// TwinCAT 3 PLC project SPS
// Company: mbc engineering GmbH
// ProgramVersion: 3.1.4022.2
// libraries:
//   Tc2_Standard, * (Beckhoff Automation GmbH)
//   Tc2_System, * (Beckhoff Automation GmbH)
//   Tc3_Module, * (Beckhoff Automation GmbH)
//   MBC TC3 PCS Library,newest,mbc engineering GmbH
// project tree:
//   Commands/ AddCommand.TcPOU, Commands.TcGVL, CustomStateCommand.TcPOU, DelayedAddCommand.TcPOU, FB_CommandWithStruct.TcPOU, PRG_Commands.TcPOU, TriggerCommand.TcPOU
//   DUTs/ E_EnumType.TcDUT, ST_CommandArgs.TcDUT
//   / PlcTask.TcTTO (not stored)
//   POUs/ MAIN.TcPOU

// ---- DUTs/E_EnumType.TcDUT
{attribute 'qualified_only'}
{attribute 'strict'}
TYPE E_EnumType :
(
	eValue0 := 0,
	eValue1 := 1,
	eValue2 := 3
);
END_TYPE

// ---- DUTs/ST_CommandArgs.TcDUT
(*
Struktur für Input-Argumente zum testen
*)
TYPE ST_CommandArgs :
STRUCT
	nNumber		: DINT;
	fFloat		: REAL;
	eEnum		: E_EnumType;
END_STRUCT
END_TYPE

// ---- Commands/Commands.TcGVL
{attribute 'qualified_only'}
VAR_GLOBAL
	fbBaseCommand1			: CommandBase;
	fbStartCommand1			: TriggerCommand;
	fbCustomStateCommand1	: CustomStateCommand;
	fbAddCommand1			: AddCommand 								:= (Val1 := 3, Val2 := 2);
	fbDelayedAddCommand1	: DelayedAddCommand(tDelayTime := T#4S) 	:= (Val1 := 10, Val2 := 4);
	fbStructCommand			: FB_CommandWithStruct;
END_VAR

// ---- Commands/TriggerCommand.TcPOU
// Command that detect the execution AND generates one cycle TRUE on the output Q
FUNCTION_BLOCK PUBLIC TriggerCommand EXTENDS CommandBase
VAR_INPUT
	bEnabled	:BOOL := TRUE;
END_VAR
VAR_OUTPUT
	Q : BOOL;
END_VAR
VAR
	bInit 	: BOOL;
END_VAR

//Enables command
stHandshake.bEnabled := bEnabled;

// OO-Class 
SUPER^();

// Will be executed in the same cycle ``stHandshake.bExecute`` changes to ``true``
METHOD PROTECTED Init
bInit := TRUE;
END_METHOD

// Execute the funktional part of the command implementation. Will be executed in the same cycle ``stHandshake.bExecute`` changes to ``true`` after the ``Init`` Method
METHOD PROTECTED Task : BOOL
// Task Code:
// dedect task completed
IF (NOT bInit AND Q) THEN
	// Task comlete;
	Task := SUPER^.Task();;
END_IF

// set output trigger
Q := bInit;

// Reset after 1. cycle
bInit := FALSE;
END_METHOD

END_FUNCTION_BLOCK

// ---- Commands/CustomStateCommand.TcPOU
FUNCTION_BLOCK CustomStateCommand EXTENDS CommandBase
VAR_INPUT
END_VAR
VAR_OUTPUT
END_VAR
VAR
	fbDelayedState: TON := (IN := FALSE, PT:= T#2S);
END_VAR

// OO-Class 
SUPER^();

// Will be called when ``stHandshake.bExecute`` changes to ``true`` one cycle and in the same cycle.
METHOD PROTECTED Init
VAR_INPUT
END_VAR
fbDelayedState(IN := False);
END_METHOD

// Execute the funktional part of the command implementation. Will also be executed in the same cycle ``stHandshake.bExecute`` changes to ``true`` after the ``Init`` Method
METHOD PROTECTED Task : BOOL

fbDelayedState(IN:= TRUE);

IF (fbDelayedState.Q) THEN
	Finish(E_CommandResultCode.StartCustom + 1);
END_IF
END_METHOD

END_FUNCTION_BLOCK

// ---- Commands/AddCommand.TcPOU
FUNCTION_BLOCK AddCommand EXTENDS CommandBase
VAR_INPUT	
END_VAR
VAR_OUTPUT		
END_VAR
VAR
	{attribute 'PlcCommandInput'}
	Val1 			: REAL;				// Value 1
	{attribute 'PlcCommandInput'}
	Val2 			: REAL;				// Value 2
	{attribute 'PlcCommandOutput'}
	Result 			: REAL;				// The result of the addition command
END_VAR

// OO-Class 
SUPER^();

METHOD PROTECTED Task : BOOL
Result := Val1 + Val2;

// Task comlete;
Task := SUPER^.Task();;
END_METHOD

END_FUNCTION_BLOCK

// ---- Commands/DelayedAddCommand.TcPOU
FUNCTION_BLOCK DelayedAddCommand EXTENDS AddCommand
VAR
	fbTonDelay		: TON;
END_VAR

// OO-Class 
SUPER^();

METHOD PROTECTED CalculateProgress
IF stHandshake.nResultCode = 99 OR stHandshake.nResultCode = E_CommandResultCode.Done THEN
	stHandshake.nProgress := 100;
ELSE
	stHandshake.nProgress := REAL_TO_BYTE(100.0 / TIME_TO_REAL(fbTonDelay.PT) * TIME_TO_REAL(fbTonDelay.ET));
END_IF
END_METHOD

METHOD Protected Cancelled
SUPER^.Cancelled();

// Reset Input for next start
fbTonDelay(IN:=stHandshake.bBusy);

// Set result to invalid value
Result := -1;
END_METHOD

METHOD PROTECTED Done
SUPER^.Done();

// Reset Input for next start
fbTonDelay(IN:=stHandshake.bBusy);
END_METHOD

METHOD FB_init : BOOL
VAR_INPUT
	bInitRetains 		: BOOL; 		// if TRUE, the retain variables are initialized (warm start / cold start)
	bInCopyCode 		: BOOL;  		// if TRUE, the instance afterwards gets moved into the copy code (online change)
	tDelayTime 			: TIME;			// Time to deleay the Running state
END_VAR
fbTonDelay.PT := tDelayTime;
END_METHOD

METHOD PROTECTED Task : BOOL
fbTonDelay(IN:=stHandshake.bBusy);

IF fbTonDelay.Q THEN
	// Execute base Task in AddCommand for Addition
	SUPER^.Task();
	
	// Exection is finished, set nResultCode = 99
	
	Finish(E_CommandResultCode.Done);
END_IF
END_METHOD

END_FUNCTION_BLOCK

// ---- Commands/FB_CommandWithStruct.TcPOU
FUNCTION_BLOCK FB_CommandWithStruct EXTENDS CommandBase
VAR
	{attribute 'PlcCommandInput'}
	stInputArgs		: ST_CommandArgs;
	{attribute 'PlcCommandInput'}
	nNumber			: INT;
	{attribute 'PlcCommandInput'}
	eEnum			: E_EnumType;
	
	{attribute 'PlcCommandOutput'}
	stOutputArgs	: ST_CommandArgs;
	{attribute 'PlcCommandOutput'}
	fFloat			: REAL;
END_VAR

SUPER^();

// Will be called when ``stHandshake.bExecute`` changes to ``true`` one cycle and in the same cycle.
METHOD PROTECTED Init
stOutputArgs := stInputArgs;
fFloat := stInputArgs.fFloat;
Finish(E_CommandResultCode.Done);
END_METHOD

END_FUNCTION_BLOCK

// ---- Commands/PRG_Commands.TcPOU
PROGRAM PRG_Commands
VAR
	fbTofStartCommand1		: TOF;		// Shows the exection was happen
END_VAR

Commands.fbBaseCommand1();
Commands.fbStartCommand1();
	
fbTofStartCommand1(
	IN := Commands.fbStartCommand1.Q,
	PT := T#2S);	
	
Commands.fbCustomStateCommand1();	
Commands.fbAddCommand1();
Commands.fbDelayedAddCommand1();
Commands.fbStructCommand();

END_PROGRAM

// ---- POUs/MAIN.TcPOU
PROGRAM MAIN
VAR
	counter				: UINT;
END_VAR

counter := counter + 1;

Commands.fbStartCommand1.bEnabled := TRUE;

PRG_Commands();

END_PROGRAM
